// TIA Portal V21 export
VAR_GLOBAL   // PLC tag table "LadderTags"
   Start AT %M26.0 : Bool;
   Stop AT %M26.1 : Bool;
   Cmd_Motor1 AT %M26.2 : Bool;
   Falha_M1 AT %M26.3 : Bool;
   Nivel_Alto AT %M26.4 : Bool;
   Auto AT %M26.5 : Bool;
   Alarme AT %M26.6 : Bool;
   Reset AT %M26.7 : Bool;
   Manutencao AT %M27.0 : Bool;
   Pronto AT %M27.1 : Bool;
   Sensor_Falha AT %M27.2 : Bool;
   Temp_OK AT %M27.3 : Bool;
   Temperatura AT %MW28 : Int;
   Setpoint AT %MW30 : Int;
END_VAR
